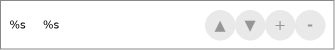
VISUALIZATION Uc_Listentry  // 335x50
    Group (0,0 335x50)
        Rectangle (0,0 335x50), colour toggle: stVisu.nSelected = nId, colour variable: Sel(bAction, colCompBg, colActionColor)
            p2167032090: colButtonDown
            OnMouseClick: execute { stVisu.nSelected := nId; }
            OnMouseDown: execute { bAction := TRUE; colActionColor := colButtonDown; }
            OnMouseEnter: execute { bAction := TRUE; colActionColor := colButtonHover; }
            OnMouseLeave: execute { bAction := FALSE; }
            OnMouseUp: execute { bAction := FALSE; }
        Group (295,10 30x30), text variable: stVisu.bRemove, invisible if: NOT (nId = stVisu.nSelected)
            OnMouseClick: execute { stVisu.nSelected := nId; stVisu.bRemove := TRUE; }
            Ellipse (0,0 30x30)
            Rectangle (0,0 30x30), "-"
        Group (265,10 30x30), text variable: stVisu.bInsert, invisible if: NOT (nId = stVisu.nSelected)
            OnMouseClick: execute { stVisu.nSelected := nId; stVisu.bInsert := TRUE; }
            Ellipse (0,0 30x30)
            Rectangle (0,0 30x30), "+"
        Group (205,10 30x30), text variable: stVisu.bInsert, invisible if: NOT (nId = stVisu.nSelected)
            OnMouseClick: execute { stVisu.nSelected := nId; stVisu.bMoveUp := TRUE; }
            Ellipse (0,0 30x30)
            Rectangle (0,0 30x30), "▲"
        Group (235,10 30x30), text variable: stVisu.bInsert, invisible if: NOT (nId = stVisu.nSelected)
            OnMouseClick: execute { stVisu.nSelected := nId; stVisu.bMoveDown := TRUE; }
            Ellipse (0,0 30x30)
            Rectangle (0,0 30x30), "▼"
        Rectangle (40,0 160x50), "%s", text variable: stVisu.astEntries[nId].sName, colour toggle: stVisu.nSelected = nId, colour variable: Sel(bAction, NormalColor, colActionColor)
            p2167032090: HighlightColor
            p3913753950: textFontName
            OnMouseClick: execute { stVisu.nSelected := nId; }
            OnMouseDown: execute { bAction := TRUE; colActionColor := colButtonDown; }
            OnMouseEnter: execute { bAction := TRUE; colActionColor := colButtonHover; }
            OnMouseLeave: execute { bAction := FALSE; }
            OnMouseUp: execute { bAction := FALSE; }
    Rectangle (0,0 35x50), "%s", text variable: nId, colour toggle: stVisu.nSelected = nId, colour variable: Sel(bAction, NormalColor, colActionColor)
        p2167032090: HighlightColor
        p3913753950: textFontName
        OnMouseClick: execute { stVisu.nSelected := nId; }
        OnMouseDown: execute { bAction := TRUE; colActionColor := colButtonDown; }
        OnMouseEnter: execute { bAction := TRUE; colActionColor := colButtonHover; }
        OnMouseLeave: execute { bAction := FALSE; }
        OnMouseUp: execute { bAction := FALSE; }
END_VISUALIZATION

(* stored: Version 1.1.0.1
   Visu Uc_Listentry: Id {dce7b4b0-2463-4e54-8501-4416d1462d2f} *)
